(* IEC 61131-3 sources: Building-Automation/HVAC System/plc, 6 files *)

(* ---- global_vars.st ---- *)
// Global Variables for HVAC Control System
// Date: June 8, 2025
// Version: 1.0.0

VAR_GLOBAL
    // System Configuration
    SYSTEM_NAME : STRING := 'HVAC Control System';
    SYSTEM_VERSION : STRING := '1.0.0';
    SCAN_TIME : TIME := T#100ms;

    // Zone Configuration
    ZONE_COUNT : INT := 8;
    ZONE_NAMES : ARRAY[1..8] OF STRING := [
        'Lobby',
        'Conference Room',
        'Office Area 1',
        'Office Area 2',
        'Kitchen',
        'Server Room',
        'Storage',
        'Break Room'
    ];

    // Temperature Control Constants
    DEFAULT_TEMP_HEATING : REAL := 21.0;     // °C
    DEFAULT_TEMP_COOLING : REAL := 24.0;     // °C
    TEMP_DEADBAND : REAL := 1.0;             // °C
    TEMP_ALARM_HIGH : REAL := 30.0;          // °C
    TEMP_ALARM_LOW : REAL := 15.0;           // °C

    // PID Control Parameters
    PID_KP : REAL := 0.8;    // Proportional gain
    PID_KI : REAL := 0.2;    // Integral gain
    PID_KD : REAL := 0.1;    // Derivative gain

    // Air Quality Constants
    CO2_SETPOINT : INT := 800;              // ppm
    CO2_ALARM_HIGH : INT := 1200;           // ppm
    HUMIDITY_SETPOINT : REAL := 50.0;       // %
    HUMIDITY_TOLERANCE : REAL := 10.0;      // %
    FRESH_AIR_MINIMUM : REAL := 15.0;       // %

    // Equipment Configuration
    SUPPLY_FAN_VFD : BOOL := TRUE;
    RETURN_FAN_VFD : BOOL := TRUE;
    COOLING_STAGES : INT := 2;
    HEATING_STAGES : INT := 2;
    ECONOMIZER_ENABLED : BOOL := TRUE;
    HEAT_RECOVERY_ENABLED : BOOL := TRUE;

    // Energy Management
    DEMAND_RESPONSE_ENABLED : BOOL := TRUE;
    PEAK_DEMAND_LIMIT : REAL := 100.0;      // kW
    OCCUPANCY_CONTROL : BOOL := TRUE;
    NIGHT_SETBACK_HEATING : REAL := 18.0;   // °C
    NIGHT_SETBACK_COOLING : REAL := 27.0;   // °C

    // Safety Parameters
    EMERGENCY_SHUTDOWN_ENABLED : BOOL := TRUE;
    FIRE_ALARM_INTEGRATION : BOOL := TRUE;
    FREEZE_PROTECTION_TEMP : REAL := 5.0;   // °C
    HIGH_TEMP_SHUTDOWN : REAL := 35.0;      // °C

    // Operating Schedule
    WEEKDAY_START : TIME_OF_DAY := TOD#07:00:00;
    WEEKDAY_END : TIME_OF_DAY := TOD#18:00:00;
    WEEKEND_START : TIME_OF_DAY := TOD#09:00:00;
    WEEKEND_END : TIME_OF_DAY := TOD#17:00:00;
    HOLIDAY_MODE : BOOL := FALSE;

    // Communication Settings
    HMI_PORT : INT := 8080;
    SIMULATOR_PORT : INT := 8081;
    MODBUS_PORT : INT := 502;
    UPDATE_INTERVAL : TIME := T#5s;

    // Maintenance Intervals
    FILTER_CHANGE_HOURS : REAL := 2160.0;   // 3 months
    BELT_INSPECTION_HOURS : REAL := 4320.0; // 6 months
    ANNUAL_MAINTENANCE_HOURS : REAL := 8760.0; // 1 year

    // Sensor Calibration Offsets
    TEMP_SENSOR_OFFSET : REAL := 0.0;
    HUMIDITY_SENSOR_OFFSET : REAL := 0.0;
    CO2_SENSOR_OFFSET : REAL := 0.0;
    PRESSURE_SENSOR_OFFSET : REAL := 0.0;

    // Runtime Data
    SYSTEM_START_TIME : DATE_AND_TIME;
    TOTAL_RUNTIME : TIME;
    ENERGY_CONSUMED : REAL;                  // kWh

    // Status Flags
    SYSTEM_INITIALIZED : BOOL := FALSE;
    FIRST_SCAN : BOOL := TRUE;
    SIMULATION_MODE : BOOL := FALSE;

END_VAR

VAR_GLOBAL CONSTANT
    // Physical Constants
    AIR_DENSITY : REAL := 1.225;           // kg/m³ at 15°C
    SPECIFIC_HEAT_AIR : REAL := 1.006;     // kJ/kg·K

    // Conversion Factors
    CFM_TO_M3S : REAL := 0.000471947;      // CFM to m³/s
    INCH_WC_TO_PA : REAL := 248.84;        // Inches of water to Pascals
    BTU_TO_KW : REAL := 0.000293071;       // BTU/hr to kW

    // Time Constants
    ONE_HOUR : TIME := T#1h;
    ONE_DAY : TIME := T#24h;
    ONE_WEEK : TIME := T#168h;

    // Equipment Limits
    MIN_FAN_SPEED : REAL := 20.0;          // %
    MAX_FAN_SPEED : REAL := 100.0;         // %
    MIN_DAMPER_POSITION : REAL := 0.0;     // %
    MAX_DAMPER_POSITION : REAL := 100.0;   // %

END_VAR

(* ---- air_quality_controller.st ---- *)
FUNCTION_BLOCK AirQualityController
VAR_INPUT
    zone_number : INT;
    co2_level : INT;           // ppm
    humidity_level : REAL;     // %
    occupancy : BOOL;
    manual_override : BOOL;
END_VAR

VAR_OUTPUT
    fresh_air_demand : REAL;   // 0-100%
    exhaust_demand : REAL;     // 0-100%
    humidity_alarm : BOOL;
    co2_alarm : BOOL;
    air_quality_fault : BOOL;
END_VAR

VAR
    co2_pid : PID;
    humidity_pid : PID;
    co2_error : REAL;
    humidity_error : REAL;

    // Alarm timers
    co2_alarm_timer : TON;
    humidity_alarm_timer : TON;

    // Demand calculation
    base_fresh_air : REAL;
    occupancy_fresh_air : REAL;
    total_fresh_air_demand : REAL;

    // Sensor fault detection
    co2_sensor_fault : BOOL;
    humidity_sensor_fault : BOOL;

    // Historical data for trending
    co2_trend : ARRAY[1..10] OF INT;
    humidity_trend : ARRAY[1..10] OF REAL;
    trend_index : INT := 1;
END_VAR

// Sensor fault detection
co2_sensor_fault := (co2_level < 300 OR co2_level > 5000);
humidity_sensor_fault := (humidity_level < 0.0 OR humidity_level > 100.0);
air_quality_fault := co2_sensor_fault OR humidity_sensor_fault;

// Update trending data
co2_trend[trend_index] := co2_level;
humidity_trend[trend_index] := humidity_level;
trend_index := trend_index + 1;
IF trend_index > 10 THEN
    trend_index := 1;
END_IF;

// CO2 Control Logic
IF NOT co2_sensor_fault THEN
    co2_error := REAL(co2_level - CO2_SETPOINT);

    // CO2 alarm detection
    co2_alarm_timer(IN := (co2_level > CO2_ALARM_HIGH), PT := T#5m);
    co2_alarm := co2_alarm_timer.Q;

    // PID control for CO2
    co2_pid(
        AUTO := TRUE,
        PV := REAL(co2_level),
        SP := REAL(CO2_SETPOINT),
        KP := 0.5,
        TI := T#600s,
        TD := T#30s,
        CYCLE := SCAN_TIME
    );

    // Calculate fresh air demand based on CO2
    IF co2_level > CO2_SETPOINT THEN
        fresh_air_demand := LIMIT(FRESH_AIR_MINIMUM, co2_pid.CV, 100.0);
    ELSE
        fresh_air_demand := FRESH_AIR_MINIMUM;
    END_IF;

ELSE
    // Sensor fault - use maximum fresh air
    fresh_air_demand := 50.0; // Conservative value
    co2_alarm := TRUE;
END_IF;

// Humidity Control Logic
IF NOT humidity_sensor_fault THEN
    humidity_error := humidity_level - HUMIDITY_SETPOINT;

    // Humidity alarm detection (high or low)
    humidity_alarm_timer(
        IN := (humidity_level > (HUMIDITY_SETPOINT + HUMIDITY_TOLERANCE) OR
               humidity_level < (HUMIDITY_SETPOINT - HUMIDITY_TOLERANCE)),
        PT := T#10m
    );
    humidity_alarm := humidity_alarm_timer.Q;

    // Humidity control through exhaust
    IF humidity_level > (HUMIDITY_SETPOINT + HUMIDITY_TOLERANCE) THEN
        exhaust_demand := LIMIT(0.0, ABS(humidity_error) * 5.0, 80.0);
    ELSE
        exhaust_demand := 0.0;
    END_IF;

ELSE
    // Sensor fault
    exhaust_demand := 0.0;
    humidity_alarm := TRUE;
END_IF;

// Occupancy-based adjustments
IF occupancy THEN
    occupancy_fresh_air := 25.0; // Higher fresh air for occupied zones
ELSE
    occupancy_fresh_air := FRESH_AIR_MINIMUM;
END_IF;

// Final fresh air demand calculation
total_fresh_air_demand := MAX(fresh_air_demand, occupancy_fresh_air);

// Manual override handling
IF manual_override THEN
    // Manual mode - maintain minimum fresh air only
    fresh_air_demand := FRESH_AIR_MINIMUM;
    exhaust_demand := 0.0;
ELSE
    fresh_air_demand := total_fresh_air_demand;
END_IF;

END_FUNCTION_BLOCK

// Main Air Quality Controller Function
FUNCTION AirQualityControllerMain : BOOL
VAR
    i : INT;
    zone_aq_controller : ARRAY[1..8] OF AirQualityController;
    total_fresh_air_demand : REAL;
    total_exhaust_demand : REAL;
    any_co2_alarm : BOOL := FALSE;
    any_humidity_alarm : BOOL := FALSE;
END_VAR

total_fresh_air_demand := 0.0;
total_exhaust_demand := 0.0;

// Process each zone
FOR i := 1 TO ZONE_COUNT DO
    zone_aq_controller[i](
        zone_number := i,
        co2_level := co2_levels[i],
        humidity_level := humidity_levels[i],
        occupancy := occupancy_detected[i],
        manual_override := FALSE
    );

    // Accumulate demands
    total_fresh_air_demand := total_fresh_air_demand + zone_aq_controller[i].fresh_air_demand;
    total_exhaust_demand := total_exhaust_demand + zone_aq_controller[i].exhaust_demand;

    // Check for any alarms
    IF zone_aq_controller[i].co2_alarm THEN
        any_co2_alarm := TRUE;
    END_IF;

    IF zone_aq_controller[i].humidity_alarm THEN
        any_humidity_alarm := TRUE;
    END_IF;
END_FOR;

// Calculate system-wide fresh air demand
outside_air_damper := LIMIT(FRESH_AIR_MINIMUM, total_fresh_air_demand / REAL(ZONE_COUNT), 100.0);

// Set global alarm flag
air_quality_alarm := any_co2_alarm OR any_humidity_alarm;

AirQualityControllerMain := TRUE;

END_FUNCTION

// Function: Air Quality Trending and Analysis
FUNCTION AirQualityTrending : BOOL
VAR
    i, j : INT;
    co2_average : REAL;
    humidity_average : REAL;
    co2_trend_slope : REAL;
    humidity_trend_slope : REAL;
END_VAR

// Calculate averages and trends for predictive control
FOR i := 1 TO ZONE_COUNT DO
    co2_average := 0.0;
    humidity_average := 0.0;

    // Calculate zone averages
    FOR j := 1 TO 10 DO
        co2_average := co2_average + REAL(co2_levels[i]);
        humidity_average := humidity_average + humidity_levels[i];
    END_FOR;

    co2_average := co2_average / 10.0;
    humidity_average := humidity_average / 10.0;

    // Predictive adjustments based on trends
    IF co2_average > (REAL(CO2_SETPOINT) * 0.9) THEN
        // Proactive fresh air increase
        outside_air_damper := outside_air_damper + 5.0;
    END_IF;
END_FOR;

AirQualityTrending := TRUE;

END_FUNCTION

// Function: Contamination Response
FUNCTION ContaminationResponse : BOOL
VAR
    i : INT;
    contamination_detected : BOOL := FALSE;
    purge_mode_active : BOOL := FALSE;
END_VAR

// Check for rapid CO2 increase (possible contamination)
FOR i := 1 TO ZONE_COUNT DO
    IF co2_levels[i] > (CO2_SETPOINT * 1.5) THEN
        contamination_detected := TRUE;
    END_IF;
END_FOR;

// Activate purge mode if contamination detected
IF contamination_detected THEN
    purge_mode_active := TRUE;
    outside_air_damper := 100.0;        // Maximum fresh air
    supply_fan_speed := 100.0;          // Maximum fan speed
    // Extend exhaust operation
END_IF;

ContaminationResponse := TRUE;

END_FUNCTION

// Function: Indoor Air Quality Index Calculation
FUNCTION CalculateIAQIndex : INT
VAR
    i : INT;
    co2_score : REAL;
    humidity_score : REAL;
    overall_score : REAL;
    zone_count_active : INT := 0;
END_VAR

overall_score := 0.0;

FOR i := 1 TO ZONE_COUNT DO
    IF occupancy_detected[i] THEN
        zone_count_active := zone_count_active + 1;

        // CO2 scoring (0-50 points)
        IF co2_levels[i] <= CO2_SETPOINT THEN
            co2_score := 50.0;
        ELSIF co2_levels[i] <= CO2_ALARM_HIGH THEN
            co2_score := 50.0 - ((REAL(co2_levels[i] - CO2_SETPOINT) / REAL(CO2_ALARM_HIGH - CO2_SETPOINT)) * 30.0);
        ELSE
            co2_score := 20.0;
        END_IF;

        // Humidity scoring (0-50 points)
        IF ABS(humidity_levels[i] - HUMIDITY_SETPOINT) <= HUMIDITY_TOLERANCE THEN
            humidity_score := 50.0;
        ELSE
            humidity_score := 50.0 - (ABS(humidity_levels[i] - HUMIDITY_SETPOINT) * 2.0);
            humidity_score := MAX(10.0, humidity_score);
        END_IF;

        overall_score := overall_score + co2_score + humidity_score;
    END_IF;
END_FOR;

IF zone_count_active > 0 THEN
    CalculateIAQIndex := REAL_TO_INT(overall_score / REAL(zone_count_active));
ELSE
    CalculateIAQIndex := 100; // Default excellent rating for unoccupied building
END_IF;

// Ensure result is within 0-100 range
CalculateIAQIndex := LIMIT(0, CalculateIAQIndex, 100);

END_FUNCTION

(* ---- energy_manager.st ---- *)
FUNCTION_BLOCK EnergyManager
VAR_INPUT
    current_demand : REAL;     // Current power demand in kW
    peak_limit : REAL;         // Peak demand limit in kW
    utility_signal : INT;      // Demand response signal (0-100)
    time_of_use_rate : REAL;   // Current electricity rate
    outside_temp : REAL;       // Outside temperature
END_VAR

VAR_OUTPUT
    demand_response_active : BOOL;
    load_shed_level : INT;     // 0-5 load shedding levels
    energy_savings_mode : BOOL;
    peak_demand_warning : BOOL;
    estimated_cost : REAL;     // Estimated hourly cost
END_VAR

VAR
    // Demand tracking
    peak_demand_today : REAL;
    peak_demand_month : REAL;
    energy_consumed_today : REAL;

    // Load shedding timers
    load_shed_timer : TON;
    recovery_timer : TON;

    // Equipment priority arrays
    equipment_priority : ARRAY[1..10] OF INT := [1,2,3,4,5,6,7,8,9,10];
    equipment_shed : ARRAY[1..10] OF BOOL;

    // Time-based controls
    current_time : TIME_OF_DAY;
    current_day : INT; // 1=Monday, 7=Sunday

    // Economic optimization
    cost_per_kwh : REAL;
    daily_energy_budget : REAL := 500.0; // kWh

    // Demand prediction
    predicted_demand : REAL;
    demand_trend : ARRAY[1..24] OF REAL; // Hourly demand history
    trend_hour : INT := 1;
END_VAR

current_time := TIME_OF_DAY();

// Update peak demand tracking
IF current_demand > peak_demand_today THEN
    peak_demand_today := current_demand;
END_IF;

IF current_demand > peak_demand_month THEN
    peak_demand_month := current_demand;
END_IF;

// Update demand trend data
demand_trend[trend_hour] := current_demand;

// Peak demand warning
peak_demand_warning := (current_demand > (peak_limit * 0.9));

// Demand response logic
IF DEMAND_RESPONSE_ENABLED THEN
    // Utility demand response signal processing
    IF utility_signal > 80 THEN
        demand_response_active := TRUE;
        load_shed_level := 4; // High demand response
    ELSIF utility_signal > 60 THEN
        demand_response_active := TRUE;
        load_shed_level := 3; // Medium demand response
    ELSIF utility_signal > 40 THEN
        demand_response_active := TRUE;
        load_shed_level := 2; // Low demand response
    ELSIF current_demand > peak_limit THEN
        demand_response_active := TRUE;
        load_shed_level := 5; // Emergency load shedding
    ELSE
        demand_response_active := FALSE;
        load_shed_level := 0; // Normal operation
    END_IF;
ELSE
    demand_response_active := FALSE;
    load_shed_level := 0;
END_IF;

// Energy savings mode activation
energy_savings_mode := (time_of_use_rate > 0.15) OR // High rate period
                      (energy_consumed_today > (daily_energy_budget * 0.8)); // Approaching budget

// Calculate estimated cost
estimated_cost := current_demand * time_of_use_rate;

// Load shedding implementation
CASE load_shed_level OF
    0: // Normal operation - no load shedding
        FOR i := 1 TO 10 DO
            equipment_shed[i] := FALSE;
        END_FOR;

    1: // Minimal load shedding - non-critical loads
        equipment_shed[1] := TRUE;  // Exterior lighting
        equipment_shed[2] := FALSE; // HVAC priority 1

    2: // Low load shedding
        equipment_shed[1] := TRUE;  // Exterior lighting
        equipment_shed[2] := TRUE;  // Non-critical HVAC zones
        equipment_shed[3] := FALSE; // Critical HVAC zones

    3: // Medium load shedding
        equipment_shed[1] := TRUE;  // Exterior lighting
        equipment_shed[2] := TRUE;  // Non-critical HVAC zones
        equipment_shed[3] := TRUE;  // Some office equipment
        equipment_shed[4] := FALSE; // Critical HVAC zones

    4: // High load shedding
        equipment_shed[1] := TRUE;  // Exterior lighting
        equipment_shed[2] := TRUE;  // Non-critical HVAC zones
        equipment_shed[3] := TRUE;  // Office equipment
        equipment_shed[4] := TRUE;  // Partial HVAC operation
        equipment_shed[5] := FALSE; // Emergency systems

    5: // Emergency load shedding
        FOR i := 1 TO 8 DO
            equipment_shed[i] := TRUE;
        END_FOR;
        equipment_shed[9] := FALSE;  // Emergency systems
        equipment_shed[10] := FALSE; // Life safety systems
END_CASE;

END_FUNCTION_BLOCK

// Main Energy Manager Function
FUNCTION EnergyManagerMain : BOOL
VAR
    energy_mgr : EnergyManager;
    current_power_demand : REAL;
    utility_dr_signal : INT;
    current_rate : REAL;

    // Equipment power consumption estimates (kW)
    supply_fan_power : REAL;
    return_fan_power : REAL;
    cooling_power : REAL;
    heating_power : REAL;
    lighting_power : REAL := 15.0;
    office_equipment_power : REAL := 25.0;
END_VAR

// Calculate equipment power consumption
supply_fan_power := (supply_fan_speed / 100.0) * 7.5; // 7.5kW max fan
return_fan_power := (return_fan_speed / 100.0) * 5.0; // 5kW max fan

IF cooling_stage_1 THEN
    cooling_power := cooling_power + 20.0; // 20kW per stage
END_IF;
IF cooling_stage_2 THEN
    cooling_power := cooling_power + 20.0;
END_IF;

IF heating_stage_1 THEN
    heating_power := heating_power + 15.0; // 15kW per stage
END_IF;
IF heating_stage_2 THEN
    heating_power := heating_power + 15.0;
END_IF;

// Total current demand
current_power_demand := supply_fan_power + return_fan_power +
                       cooling_power + heating_power +
                       lighting_power + office_equipment_power;

// Get time-of-use rate (simplified)
IF current_time >= TOD#08:00:00 AND current_time <= TOD#20:00:00 THEN
    current_rate := 0.18; // Peak rate
ELSE
    current_rate := 0.12; // Off-peak rate
END_IF;

// Simulate utility demand response signal
utility_dr_signal := 0; // Normal operation

// Run energy manager
energy_mgr(
    current_demand := current_power_demand,
    peak_limit := PEAK_DEMAND_LIMIT,
    utility_signal := utility_dr_signal,
    time_of_use_rate := current_rate,
    outside_temp := outdoor_temp
);

// Apply load shedding actions
ApplyLoadShedding(energy_mgr.load_shed_level);

// Update global energy management flags
demand_response_active := energy_mgr.demand_response_active;

EnergyManagerMain := TRUE;

END_FUNCTION

// Function: Apply Load Shedding
FUNCTION ApplyLoadShedding : BOOL
VAR_INPUT
    shed_level : INT;
END_VAR
VAR
    temp_setpoint_offset : REAL;
    fan_speed_reduction : REAL;
END_VAR

CASE shed_level OF
    0: // Normal operation
        temp_setpoint_offset := 0.0;
        fan_speed_reduction := 0.0;

    1: // Minimal shedding
        temp_setpoint_offset := 0.5; // Slight setpoint adjustment
        fan_speed_reduction := 5.0;  // 5% fan speed reduction

    2: // Low shedding
        temp_setpoint_offset := 1.0;
        fan_speed_reduction := 10.0;

    3: // Medium shedding
        temp_setpoint_offset := 1.5;
        fan_speed_reduction := 15.0;

    4: // High shedding
        temp_setpoint_offset := 2.0;
        fan_speed_reduction := 20.0;

    5: // Emergency shedding
        temp_setpoint_offset := 3.0;
        fan_speed_reduction := 30.0;
END_CASE;

// Apply temperature setpoint adjustments
FOR i := 1 TO ZONE_COUNT DO
    IF zone_heating_demand[i] THEN
        zone_setpoints[i] := zone_setpoints[i] - temp_setpoint_offset;
    ELSIF zone_cooling_demand[i] THEN
        zone_setpoints[i] := zone_setpoints[i] + temp_setpoint_offset;
    END_IF;
END_FOR;

// Apply fan speed reduction
supply_fan_speed := supply_fan_speed * (1.0 - fan_speed_reduction / 100.0);
return_fan_speed := return_fan_speed * (1.0 - fan_speed_reduction / 100.0);

// Limit minimum values
supply_fan_speed := MAX(MIN_FAN_SPEED, supply_fan_speed);
return_fan_speed := MAX(MIN_FAN_SPEED, return_fan_speed);

ApplyLoadShedding := TRUE;

END_FUNCTION

// Function: Optimal Start/Stop Control
FUNCTION OptimalStartStop : BOOL
VAR
    building_thermal_mass : REAL := 2.5; // Hours to change 1°C
    preheat_time : TIME;
    precool_time : TIME;
    start_time : TIME_OF_DAY;
    stop_time : TIME_OF_DAY;
    temp_difference : REAL;
END_VAR

// Calculate required pre-conditioning time
IF outdoor_temp < 15.0 THEN
    // Heating season
    temp_difference := DEFAULT_TEMP_HEATING - 18.0; // Night setback difference
    preheat_time := REAL_TO_TIME(REAL_TO_DINT(temp_difference * building_thermal_mass * 3600000.0));

    // Adjust start time for optimal pre-heating
    start_time := WEEKDAY_START - TIME_TO_TOD(preheat_time);

ELSIF outdoor_temp > 25.0 THEN
    // Cooling season
    temp_difference := 27.0 - DEFAULT_TEMP_COOLING; // Night setback difference
    precool_time := REAL_TO_TIME(REAL_TO_DINT(temp_difference * building_thermal_mass * 3600000.0));

    // Adjust start time for optimal pre-cooling
    start_time := WEEKDAY_START - TIME_TO_TOD(precool_time);
ELSE
    // Mild weather - normal start time
    start_time := WEEKDAY_START;
END_IF;

// Optimal stop control with thermal flywheel
stop_time := WEEKDAY_END - T#30m; // Stop 30 minutes early

OptimalStartStop := TRUE;

END_FUNCTION

// Function: Energy Reporting
FUNCTION EnergyReporting : BOOL
VAR
    daily_consumption : REAL;
    monthly_consumption : REAL;
    energy_efficiency_ratio : REAL;
    carbon_footprint : REAL;
    cost_savings : REAL;
END_VAR

// Calculate energy efficiency metrics
energy_efficiency_ratio := daily_consumption / (outdoor_temp * 24.0); // Simplified EER

// Calculate carbon footprint (kg CO2)
carbon_footprint := daily_consumption * 0.45; // 0.45 kg CO2/kWh average

// Calculate cost savings from demand response
cost_savings := 0.0; // Calculate based on load shedding actions

EnergyReporting := TRUE;

END_FUNCTION

(* ---- safety_controller.st ---- *)
FUNCTION_BLOCK SafetyController
VAR_INPUT
    fire_alarm_input : BOOL;
    smoke_detector : ARRAY[1..8] OF BOOL;
    freeze_stat : BOOL;
    high_pressure_alarm : BOOL;
    low_pressure_alarm : BOOL;
    manual_emergency_stop : BOOL;
END_VAR

VAR_OUTPUT
    emergency_shutdown : BOOL;
    fire_mode_active : BOOL;
    freeze_protection_active : BOOL;
    safety_fault : BOOL;
    smoke_purge_active : BOOL;
END_VAR

VAR
    // Safety timers
    fire_alarm_timer : TON;
    freeze_protection_timer : TON;
    smoke_purge_timer : TON;

    // Safety status tracking
    any_smoke_detected : BOOL;
    freeze_protection_required : BOOL;
    pressure_fault : BOOL;

    // Safety interlocks
    supply_fan_safety : BOOL;
    return_fan_safety : BOOL;
    outside_air_safety : BOOL;

    // Emergency sequences
    fire_sequence_step : INT;
    freeze_sequence_step : INT;

    // Safety override flags
    manual_override_active : BOOL;
    maintenance_mode : BOOL;
END_VAR

// Smoke detection logic
any_smoke_detected := FALSE;
FOR i := 1 TO 8 DO
    IF smoke_detector[i] THEN
        any_smoke_detected := TRUE;
    END_IF;
END_FOR;

// Fire alarm processing with confirmation timer
fire_alarm_timer(IN := (fire_alarm_input OR any_smoke_detected), PT := T#5s);
fire_mode_active := fire_alarm_timer.Q;

// Freeze protection logic
freeze_protection_required := (outdoor_temp <= FREEZE_PROTECTION_TEMP) OR freeze_stat;
freeze_protection_timer(IN := freeze_protection_required, PT := T#10s);
freeze_protection_active := freeze_protection_timer.Q;

// Pressure fault detection
pressure_fault := high_pressure_alarm OR low_pressure_alarm;

// Main safety fault logic
safety_fault := pressure_fault OR manual_emergency_stop;

// Emergency shutdown conditions
emergency_shutdown := fire_mode_active OR
                     freeze_protection_active OR
                     safety_fault OR
                     (outdoor_temp > HIGH_TEMP_SHUTDOWN);

// Smoke purge sequence
IF any_smoke_detected AND NOT fire_mode_active THEN
    smoke_purge_timer(IN := TRUE, PT := T#10m);
    smoke_purge_active := smoke_purge_timer.Q;
ELSE
    smoke_purge_timer(IN := FALSE);
    smoke_purge_active := FALSE;
END_IF;

// Safety interlocks for equipment
supply_fan_safety := NOT emergency_shutdown;
return_fan_safety := NOT emergency_shutdown;
outside_air_safety := NOT (fire_mode_active OR freeze_protection_active);

END_FUNCTION_BLOCK

// Main Safety Controller Function
FUNCTION SafetyControllerMain : BOOL
VAR
    safety_ctrl : SafetyController;
    i : INT;
    any_zone_overtemp : BOOL := FALSE;
    any_zone_undertemp : BOOL := FALSE;
END_VAR

// Check for temperature safety conditions
FOR i := 1 TO ZONE_COUNT DO
    IF zone_temps[i] > TEMP_ALARM_HIGH THEN
        any_zone_overtemp := TRUE;
    END_IF;

    IF zone_temps[i] < TEMP_ALARM_LOW THEN
        any_zone_undertemp := TRUE;
    END_IF;
END_FOR;

// Run main safety controller
safety_ctrl(
    fire_alarm_input := fire_alarm,
    smoke_detector := smoke_detector,
    freeze_stat := (outdoor_temp <= FREEZE_PROTECTION_TEMP),
    high_pressure_alarm := FALSE, // Connect to actual pressure sensors
    low_pressure_alarm := FALSE,  // Connect to actual pressure sensors
    manual_emergency_stop := emergency_stop
);

// Update global safety flags
emergency_stop := safety_ctrl.emergency_shutdown;
fire_mode_active := safety_ctrl.fire_mode_active;
freeze_protection_active := safety_ctrl.freeze_protection_active;
system_fault := safety_ctrl.safety_fault;

// Implement safety actions
IF safety_ctrl.fire_mode_active THEN
    FireModeSequence();
END_IF;

IF safety_ctrl.freeze_protection_active THEN
    FreezeProtectionSequence();
END_IF;

IF safety_ctrl.smoke_purge_active THEN
    SmokePurgeSequence();
END_IF;

SafetyControllerMain := TRUE;

END_FUNCTION

// Function: Fire Mode Sequence
FUNCTION FireModeSequence : BOOL
VAR
    fire_sequence_timer : TON;
END_VAR

// Fire mode operation sequence according to NFPA standards
// 1. Shut down return fans immediately
return_fan_running := FALSE;
return_fan_speed := 0.0;

// 2. Close outside air dampers
outside_air_damper := 0.0;

// 3. Stop heating and cooling
heating_stage_1 := FALSE;
heating_stage_2 := FALSE;
cooling_stage_1 := FALSE;
cooling_stage_2 := FALSE;

// 4. Supply fan operation depends on fire department connection
// For pressurization mode, keep supply fan running at low speed
IF fire_alarm THEN
    supply_fan_running := TRUE;
    supply_fan_speed := 30.0; // Low speed for stairwell pressurization
ELSE
    supply_fan_running := FALSE;
    supply_fan_speed := 0.0;
END_IF;

// 5. Activate building management system notifications
// (This would interface with BMS)

FireModeSequence := TRUE;

END_FUNCTION

// Function: Freeze Protection Sequence
FUNCTION FreezeProtectionSequence : BOOL
VAR
    freeze_timer : TON;
END_VAR

// Freeze protection sequence
// 1. Close outside air damper to minimum
outside_air_damper := 0.0;

// 2. Start supply fan for air circulation
supply_fan_running := TRUE;
supply_fan_speed := 50.0; // Moderate speed for circulation

// 3. Start return fan
return_fan_running := TRUE;
return_fan_speed := 50.0;

// 4. Activate heating if available
heating_stage_1 := TRUE;
IF outdoor_temp <= (FREEZE_PROTECTION_TEMP - 2.0) THEN
    heating_stage_2 := TRUE;
END_IF;

// 5. Disable cooling
cooling_stage_1 := FALSE;
cooling_stage_2 := FALSE;

// 6. Override temperature setpoints to prevent freezing
FOR i := 1 TO ZONE_COUNT DO
    zone_setpoints[i] := MAX(zone_setpoints[i], 10.0);
END_FOR;

FreezeProtectionSequence := TRUE;

END_FUNCTION

// Function: Smoke Purge Sequence
FUNCTION SmokePurgeSequence : BOOL
VAR
    purge_timer : TON;
END_VAR

// Smoke purge sequence (not fire mode)
// 1. Increase outside air to maximum
outside_air_damper := 100.0;

// 2. Run fans at high speed
supply_fan_running := TRUE;
supply_fan_speed := 100.0;
return_fan_running := TRUE;
return_fan_speed := 100.0;

// 3. Disable heating and cooling during purge
heating_stage_1 := FALSE;
heating_stage_2 := FALSE;
cooling_stage_1 := FALSE;
cooling_stage_2 := FALSE;

// 4. Continue purge for specified time (10 minutes)
purge_timer(IN := TRUE, PT := T#10m);

// 5. Return to normal operation after purge
IF purge_timer.Q THEN
    smoke_purge_active := FALSE;
END_IF;

SmokePurgeSequence := TRUE;

END_FUNCTION

// Function: Safety System Test
FUNCTION SafetySystemTest : BOOL
VAR
    test_sequence_step : INT;
    test_timer : TON;
    test_results : ARRAY[1..10] OF BOOL;
END_VAR

// Weekly automatic safety system test
// This function would be called during maintenance windows

CASE test_sequence_step OF
    0: // Initialize test
        test_sequence_step := 1;

    1: // Test smoke detectors
        // Simulate smoke detection test
        test_timer(IN := TRUE, PT := T#30s);
        IF test_timer.Q THEN
            test_results[1] := TRUE; // Test passed
            test_sequence_step := 2;
            test_timer(IN := FALSE);
        END_IF;

    2: // Test fire alarm interface
        test_timer(IN := TRUE, PT := T#30s);
        IF test_timer.Q THEN
            test_results[2] := TRUE;
            test_sequence_step := 3;
            test_timer(IN := FALSE);
        END_IF;

    3: // Test freeze protection
        test_timer(IN := TRUE, PT := T#30s);
        IF test_timer.Q THEN
            test_results[3] := TRUE;
            test_sequence_step := 4;
            test_timer(IN := FALSE);
        END_IF;

    4: // Test emergency stop
        test_timer(IN := TRUE, PT := T#30s);
        IF test_timer.Q THEN
            test_results[4] := TRUE;
            test_sequence_step := 0; // Test complete
            test_timer(IN := FALSE);
        END_IF;
END_CASE;

SafetySystemTest := TRUE;

END_FUNCTION

// Function: Safety Alarm Prioritization
FUNCTION SafetyAlarmPriority : INT
VAR
    priority_level : INT;
END_VAR

// Determine highest priority safety alarm
IF fire_alarm THEN
    priority_level := 1; // Highest priority
ELSIF emergency_stop THEN
    priority_level := 2;
ELSIF freeze_protection_active THEN
    priority_level := 3;
ELSIF high_temp_alarm THEN
    priority_level := 4;
ELSIF air_quality_alarm THEN
    priority_level := 5;
ELSE
    priority_level := 0; // No alarms
END_IF;

SafetyAlarmPriority := priority_level;

END_FUNCTION

// Function: Safety Interlock Check
FUNCTION SafetyInterlockCheck : BOOL
VAR
    interlock_ok : BOOL := TRUE;
END_VAR

// Check all safety interlocks before starting equipment

// Check fire safety
IF fire_mode_active THEN
    interlock_ok := FALSE;
END_IF;

// Check freeze protection
IF freeze_protection_active AND outside_air_damper > 10.0 THEN
    interlock_ok := FALSE;
END_IF;

// Check pressure safety
IF high_pressure_alarm OR low_pressure_alarm THEN
    interlock_ok := FALSE;
END_IF;

// Check temperature limits
FOR i := 1 TO ZONE_COUNT DO
    IF zone_temps[i] > HIGH_TEMP_SHUTDOWN OR zone_temps[i] < FREEZE_PROTECTION_TEMP THEN
        interlock_ok := FALSE;
    END_IF;
END_FOR;

SafetyInterlockCheck := interlock_ok;

END_FUNCTION

(* ---- temperature_controller.st ---- *)
FUNCTION_BLOCK TemperatureController
VAR_INPUT
    zone_number : INT;
    current_temp : REAL;
    setpoint_heating : REAL;
    setpoint_cooling : REAL;
    occupancy : BOOL;
    manual_override : BOOL;
END_VAR

VAR_OUTPUT
    heating_demand : BOOL;
    cooling_demand : BOOL;
    demand_level : REAL; // 0.0 to 1.0
    zone_fault : BOOL;
END_VAR

VAR
    pid_heating : PID;
    pid_cooling : PID;
    temp_error : REAL;
    deadband_high : REAL;
    deadband_low : REAL;
    last_temp : REAL;
    temp_change_rate : REAL;
    alarm_timer : TON;
    fault_timer : TON;

    // Night setback variables
    effective_setpoint_heating : REAL;
    effective_setpoint_cooling : REAL;

    // Alarm conditions
    high_temp_alarm : BOOL;
    low_temp_alarm : BOOL;
    sensor_fault : BOOL;
END_VAR

// Calculate effective setpoints (considering night setback)
IF NOT occupancy AND NOT manual_override THEN
    effective_setpoint_heating := NIGHT_SETBACK_HEATING;
    effective_setpoint_cooling := NIGHT_SETBACK_COOLING;
ELSE
    effective_setpoint_heating := setpoint_heating;
    effective_setpoint_cooling := setpoint_cooling;
END_IF;

// Calculate deadband limits
deadband_low := effective_setpoint_heating - (TEMP_DEADBAND / 2.0);
deadband_high := effective_setpoint_cooling + (TEMP_DEADBAND / 2.0);

// Temperature change rate calculation
temp_change_rate := (current_temp - last_temp) / (TIME_TO_REAL(SCAN_TIME) / 1000.0);
last_temp := current_temp;

// Sensor fault detection
IF current_temp < -50.0 OR current_temp > 80.0 THEN
    sensor_fault := TRUE;
ELSE
    sensor_fault := FALSE;
END_IF;

// Temperature alarm detection
high_temp_alarm := current_temp > TEMP_ALARM_HIGH;
low_temp_alarm := current_temp < TEMP_ALARM_LOW;

// Fault timer for persistent alarms
fault_timer(IN := (high_temp_alarm OR low_temp_alarm OR sensor_fault), PT := T#30s);
zone_fault := fault_timer.Q;

// Main control logic (only if no sensor fault)
IF NOT sensor_fault THEN

    // Heating Control
    IF current_temp < deadband_low THEN
        heating_demand := TRUE;
        cooling_demand := FALSE;

        // PID control for heating
        pid_heating(
            AUTO := TRUE,
            PV := current_temp,
            SP := effective_setpoint_heating,
            KP := PID_KP,
            TI := T#300s,
            TD := T#60s,
            CYCLE := SCAN_TIME
        );

        demand_level := LIMIT(0.0, pid_heating.CV / 100.0, 1.0);

    // Cooling Control
    ELSIF current_temp > deadband_high THEN
        cooling_demand := TRUE;
        heating_demand := FALSE;

        // PID control for cooling
        pid_cooling(
            AUTO := TRUE,
            PV := current_temp,
            SP := effective_setpoint_cooling,
            KP := PID_KP,
            TI := T#300s,
            TD := T#60s,
            CYCLE := SCAN_TIME
        );

        demand_level := LIMIT(0.0, pid_cooling.CV / 100.0, 1.0);

    // Dead band - no heating or cooling
    ELSE
        heating_demand := FALSE;
        cooling_demand := FALSE;
        demand_level := 0.0;

        // Reset PID controllers
        pid_heating(AUTO := FALSE);
        pid_cooling(AUTO := FALSE);
    END_IF;

ELSE
    // Sensor fault - safe mode
    heating_demand := FALSE;
    cooling_demand := FALSE;
    demand_level := 0.0;
END_IF;

END_FUNCTION_BLOCK

// Main Temperature Controller Function
FUNCTION TemperatureControllerMain : BOOL
VAR
    i : INT;
    zone_controller : ARRAY[1..8] OF TemperatureController;
    total_heating_demand : INT := 0;
    total_cooling_demand : INT := 0;
END_VAR

// Process each zone
FOR i := 1 TO ZONE_COUNT DO
    zone_controller[i](
        zone_number := i,
        current_temp := zone_temps[i],
        setpoint_heating := zone_setpoints[i],
        setpoint_cooling := zone_setpoints[i] + 3.0, // 3°C cooling offset
        occupancy := occupancy_detected[i],
        manual_override := FALSE
    );

    // Update global arrays
    zone_heating_demand[i] := zone_controller[i].heating_demand;
    zone_cooling_demand[i] := zone_controller[i].cooling_demand;

    // Count total demands
    IF zone_controller[i].heating_demand THEN
        total_heating_demand := total_heating_demand + 1;
    END_IF;

    IF zone_controller[i].cooling_demand THEN
        total_cooling_demand := total_cooling_demand + 1;
    END_IF;
END_FOR;

// Update system demand indicators
any_heating_demand := total_heating_demand > 0;
any_cooling_demand := total_cooling_demand > 0;

TemperatureControllerMain := TRUE;

END_FUNCTION

// Function: Initialize Zone Setpoints
FUNCTION InitializeZoneSetpoints : BOOL
VAR
    i : INT;
END_VAR

FOR i := 1 TO ZONE_COUNT DO
    CASE i OF
        1: zone_setpoints[i] := 22.0; // Lobby
        2: zone_setpoints[i] := 23.0; // Conference Room
        3, 4: zone_setpoints[i] := 22.0; // Office Areas
        5: zone_setpoints[i] := 21.0; // Kitchen
        6: zone_setpoints[i] := 20.0; // Server Room (cooler)
        7: zone_setpoints[i] := 18.0; // Storage (minimal heating)
        8: zone_setpoints[i] := 22.0; // Break Room
    ELSE
        zone_setpoints[i] := DEFAULT_TEMP_HEATING;
    END_CASE;
END_FOR;

InitializeZoneSetpoints := TRUE;

END_FUNCTION

// Function: Adaptive Temperature Control
FUNCTION AdaptiveTempControl : BOOL
VAR
    i : INT;
    outdoor_temp_factor : REAL;
    occupancy_factor : REAL;
    time_of_day : TIME_OF_DAY;
END_VAR

time_of_day := TIME_OF_DAY();

// Adjust setpoints based on outdoor temperature
IF outdoor_temp < 0.0 THEN
    outdoor_temp_factor := 1.0; // Colder setpoint offset
ELSIF outdoor_temp > 30.0 THEN
    outdoor_temp_factor := -1.0; // Warmer setpoint offset
ELSE
    outdoor_temp_factor := 0.0; // No adjustment
END_IF;

// Adjust setpoints based on time of day and occupancy
FOR i := 1 TO ZONE_COUNT DO
    // Morning warm-up
    IF time_of_day >= TOD#06:00:00 AND time_of_day <= TOD#08:00:00 THEN
        zone_setpoints[i] := zone_setpoints[i] + 1.0;
    END_IF;

    // Afternoon adjustment
    IF time_of_day >= TOD#14:00:00 AND time_of_day <= TOD#16:00:00 THEN
        zone_setpoints[i] := zone_setpoints[i] - 0.5;
    END_IF;

    // Apply outdoor temperature compensation
    zone_setpoints[i] := zone_setpoints[i] + outdoor_temp_factor;

    // Limit setpoint ranges
    zone_setpoints[i] := LIMIT(18.0, zone_setpoints[i], 26.0);
END_FOR;

AdaptiveTempControl := TRUE;

END_FUNCTION

(* ---- main.st ---- *)
PROGRAM Main
VAR
    // System Status Variables
    system_running : BOOL := FALSE;
    emergency_stop : BOOL := FALSE;
    system_fault : BOOL := FALSE;

    // Temperature Control
    zone_temps : ARRAY[1..8] OF REAL;
    zone_setpoints : ARRAY[1..8] OF REAL;
    zone_heating_demand : ARRAY[1..8] OF BOOL;
    zone_cooling_demand : ARRAY[1..8] OF BOOL;

    // Air Quality
    co2_levels : ARRAY[1..8] OF INT;
    humidity_levels : ARRAY[1..8] OF REAL;
    air_quality_alarm : BOOL := FALSE;

    // Equipment Status
    supply_fan_running : BOOL := FALSE;
    return_fan_running : BOOL := FALSE;
    cooling_stage_1 : BOOL := FALSE;
    cooling_stage_2 : BOOL := FALSE;
    heating_stage_1 : BOOL := FALSE;
    heating_stage_2 : BOOL := FALSE;
    economizer_active : BOOL := FALSE;

    // Safety Systems
    fire_alarm : BOOL := FALSE;
    freeze_protection_active : BOOL := FALSE;
    high_temp_alarm : BOOL := FALSE;

    // Energy Management
    demand_response_active : BOOL := FALSE;
    night_setback_active : BOOL := FALSE;
    occupancy_detected : ARRAY[1..8] OF BOOL;

    // Timers
    system_runtime : TIME;
    filter_runtime : TIME;
    maintenance_timer : TIME;

    // Control Variables
    outdoor_temp : REAL;
    outdoor_humidity : REAL;
    outside_air_damper : REAL; // 0-100%
    supply_fan_speed : REAL; // 0-100%
    return_fan_speed : REAL; // 0-100%

    // Maintenance
    filter_change_required : BOOL := FALSE;
    maintenance_required : BOOL := FALSE;

    // Communication
    hmi_connected : BOOL := FALSE;
    data_logging_active : BOOL := FALSE;
END_VAR

// Main Program Logic
IF NOT emergency_stop AND NOT system_fault THEN
    system_running := TRUE;

    // Call Temperature Controller
    TemperatureController();

    // Call Air Quality Controller
    AirQualityController();

    // Call Energy Manager
    EnergyManager();

    // Call Safety Controller
    SafetyController();

    // Update Equipment Status
    UpdateEquipmentStatus();

    // Handle Maintenance Checks
    MaintenanceCheck();

ELSE
    // Emergency shutdown sequence
    EmergencyShutdown();
    system_running := FALSE;
END_IF;

// Always run communication regardless of system status
CommunicationHandler();

END_PROGRAM

// Function: Update Equipment Status
FUNCTION UpdateEquipmentStatus : BOOL
VAR
    any_heating_demand : BOOL := FALSE;
    any_cooling_demand : BOOL := FALSE;
    total_demand : REAL;
    i : INT;
END_VAR

// Check for any zone demands
FOR i := 1 TO 8 DO
    IF zone_heating_demand[i] THEN
        any_heating_demand := TRUE;
    END_IF;
    IF zone_cooling_demand[i] THEN
        any_cooling_demand := TRUE;
    END_IF;
END_FOR;

// Supply Fan Control
IF system_running AND (any_heating_demand OR any_cooling_demand OR economizer_active) THEN
    supply_fan_running := TRUE;
    // Calculate fan speed based on demand
    supply_fan_speed := MAX(30.0, MIN(100.0, total_demand * 50.0 + 30.0));
ELSE
    supply_fan_running := FALSE;
    supply_fan_speed := 0.0;
END_IF;

// Return Fan Control
return_fan_running := supply_fan_running;
return_fan_speed := supply_fan_speed * 0.9; // 90% of supply fan speed

// Heating Control
IF any_heating_demand AND system_running THEN
    heating_stage_1 := TRUE;
    // Stage 2 heating if high demand
    IF total_demand > 0.7 THEN
        heating_stage_2 := TRUE;
    ELSE
        heating_stage_2 := FALSE;
    END_IF;
ELSE
    heating_stage_1 := FALSE;
    heating_stage_2 := FALSE;
END_IF;

// Cooling Control
IF any_cooling_demand AND system_running THEN
    cooling_stage_1 := TRUE;
    // Stage 2 cooling if high demand
    IF total_demand > 0.7 THEN
        cooling_stage_2 := TRUE;
    ELSE
        cooling_stage_2 := FALSE;
    END_IF;
ELSE
    cooling_stage_1 := FALSE;
    cooling_stage_2 := FALSE;
END_IF;

// Economizer Control
IF system_running AND outdoor_temp < 18.0 AND any_cooling_demand THEN
    economizer_active := TRUE;
    outside_air_damper := MIN(100.0, total_demand * 80.0);
ELSE
    economizer_active := FALSE;
    outside_air_damper := 15.0; // Minimum fresh air
END_IF;

UpdateEquipmentStatus := TRUE;

END_FUNCTION

// Function: Emergency Shutdown
FUNCTION EmergencyShutdown : BOOL
VAR
END_VAR

// Shut down all equipment immediately
supply_fan_running := FALSE;
return_fan_running := FALSE;
heating_stage_1 := FALSE;
heating_stage_2 := FALSE;
cooling_stage_1 := FALSE;
cooling_stage_2 := FALSE;
economizer_active := FALSE;

// Close dampers
outside_air_damper := 0.0;

// Set all outputs to safe state
supply_fan_speed := 0.0;
return_fan_speed := 0.0;

EmergencyShutdown := TRUE;

END_FUNCTION

// Function: Maintenance Check
FUNCTION MaintenanceCheck : BOOL
VAR
    filter_hours : REAL;
    maintenance_hours : REAL;
END_VAR

// Convert runtime to hours
filter_hours := TIME_TO_REAL(filter_runtime) / 3600000.0; // Convert ms to hours
maintenance_hours := TIME_TO_REAL(maintenance_timer) / 3600000.0;

// Check filter replacement
IF filter_hours >= 2160.0 THEN // 3 months
    filter_change_required := TRUE;
END_IF;

// Check maintenance schedule
IF maintenance_hours >= 8760.0 THEN // 1 year
    maintenance_required := TRUE;
END_IF;

MaintenanceCheck := TRUE;

END_FUNCTION

// Function: Communication Handler
FUNCTION CommunicationHandler : BOOL
VAR
END_VAR

// Update HMI data
// This would interface with the HMI system
// Update data logging
// This would handle data logging functions

// Check for commands from HMI
// Process setpoint changes, schedule updates, etc.

CommunicationHandler := TRUE;

END_FUNCTION
